FUNCTION_BLOCK fb_motorController
VAR_INPUT
	in_flg_run : BOOL;
END_VAR
VAR_OUTPUT
	out_flg_run : bool;
END_VAR
VAR
	flg_mototPowerRun: BOOL;
	flg_motorPowerReset: bool;
	fbi_delayTimerY: TON;
	fbi_delayTimerZ: TON;
	flg_rotaryPowerRun: BOOL;
	fbi_delayTimer1: TON;
END_VAR
VAR // added by the converter: edge detectors and wires of the graphical bodies
    _rt1, _rt2, _rt3, _rt4, _rt5, _rt6 : R_TRIG;
    _ft1, _ft2 : F_TRIG;
END_VAR

motorPower();
motorMoveAbs();
gm_rotary();
IF  gvl_param.var_currentMode = eP_programMode.manual OR gvl_param.var_currentMode = eP_programMode.error THEN
	motorJog();
END_IF
IF gvl_axis.axisX.NcToPlc.ActTorque > 500 THEN
	gvl_error.flg_axisXTorqueOver := TRUE;
ELSIF gvl_axis.axisY.NcToPlc.ActTorque > 500 THEN
	gvl_error.flg_axisYTorqueOver := TRUE;
ELSIF gvl_axis.axisZ.NcToPlc.ActTorque > 500 THEN
	gvl_error.flg_axisZTorqueOver := TRUE;
ELSIF gvl_axis.axisR.NcToPlc.ActTorque > 500 THEN
	gvl_error.flg_axisRTorqueOver := TRUE;
ELSE
	gvl_error.flg_axisXTorqueOver := FALSE;
	gvl_error.flg_axisYTorqueOver := FALSE;
	gvl_error.flg_axisZTorqueOver := FALSE;
	gvl_error.flg_axisRTorqueOver := FALSE;
END_IF

ACTION gm_rotary:
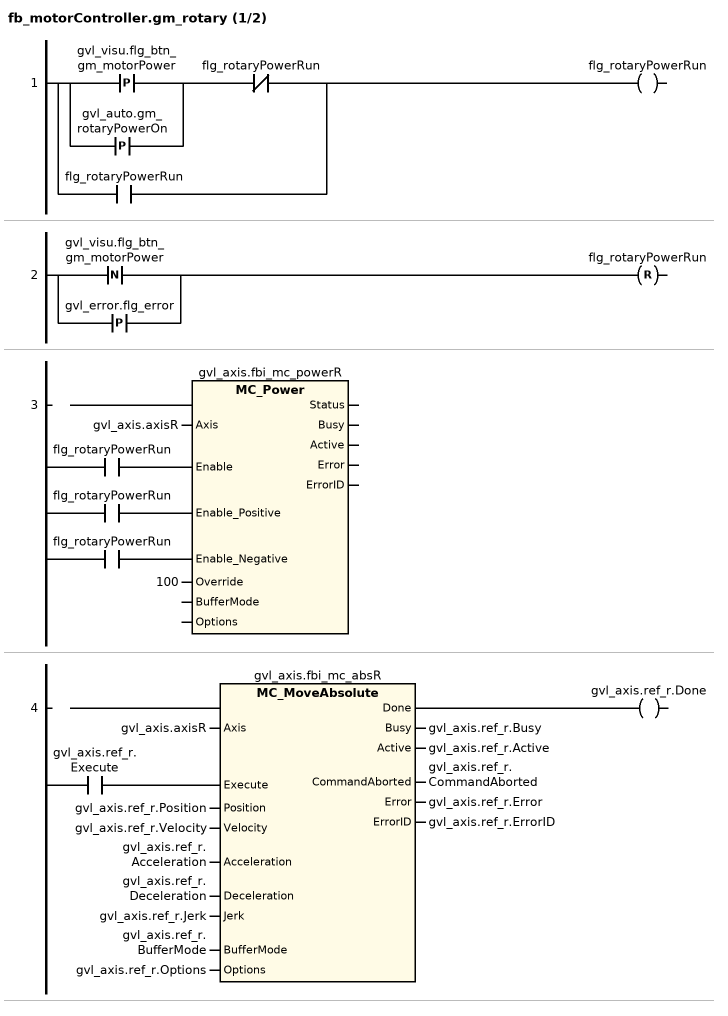
// NETWORK 1
_rt1(CLK := gvl_visu.flg_btn_gm_motorPower);
_rt2(CLK := gvl_auto.gm_rotaryPowerOn);
flg_rotaryPowerRun := (_rt1.Q OR _rt2.Q) AND NOT flg_rotaryPowerRun OR flg_rotaryPowerRun;

// NETWORK 2
_ft1(CLK := gvl_visu.flg_btn_gm_motorPower);
_rt3(CLK := gvl_error.flg_error);
flg_rotaryPowerRun R= _ft1.Q OR _rt3.Q;

// NETWORK 3
gvl_axis.fbi_mc_powerR(
    Axis := gvl_axis.axisR,
    Enable := flg_rotaryPowerRun,
    Enable_Positive := flg_rotaryPowerRun,
    Enable_Negative := flg_rotaryPowerRun,
    Override := 100); // MC_Power

// NETWORK 4
gvl_axis.fbi_mc_absR(
    Axis := gvl_axis.axisR,
    Execute := gvl_axis.ref_r.Execute,
    Position := gvl_axis.ref_r.Position,
    Velocity := gvl_axis.ref_r.Velocity,
    Acceleration := gvl_axis.ref_r.Acceleration,
    Deceleration := gvl_axis.ref_r.Deceleration,
    Jerk := gvl_axis.ref_r.Jerk,
    BufferMode := gvl_axis.ref_r.BufferMode,
    Options := gvl_axis.ref_r.Options,
    Busy => gvl_axis.ref_r.Busy,
    Active => gvl_axis.ref_r.Active,
    CommandAborted => gvl_axis.ref_r.CommandAborted,
    Error => gvl_axis.ref_r.Error,
    ErrorID => gvl_axis.ref_r.ErrorID); // MC_MoveAbsolute
gvl_axis.ref_r.Done := gvl_axis.fbi_mc_absR.Done;

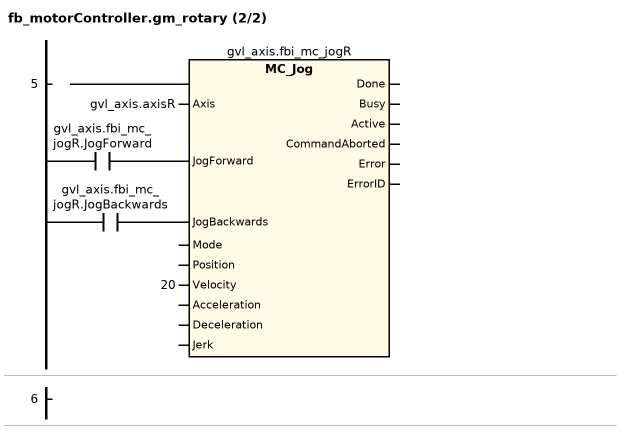
// NETWORK 5
gvl_axis.fbi_mc_jogR(
    Axis := gvl_axis.axisR,
    JogForward := gvl_axis.fbi_mc_jogR.JogForward,
    JogBackwards := gvl_axis.fbi_mc_jogR.JogBackwards,
    Velocity := 20); // MC_Jog

// NETWORK 6
END_ACTION

ACTION motorJog:
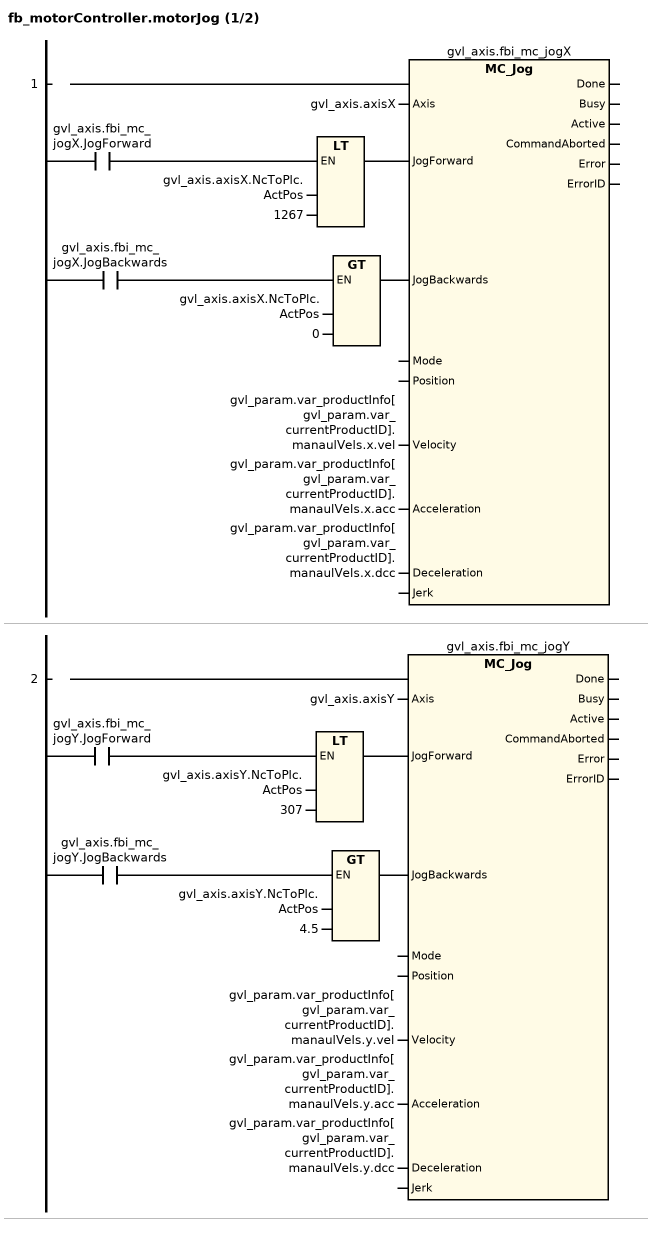
// NETWORK 1
gvl_axis.fbi_mc_jogX(
    Axis := gvl_axis.axisX,
    JogForward := gvl_axis.fbi_mc_jogX.JogForward AND gvl_axis.axisX.NcToPlc.ActPos < 1267,
    JogBackwards := gvl_axis.fbi_mc_jogX.JogBackwards AND gvl_axis.axisX.NcToPlc.ActPos > 0,
    Velocity := gvl_param.var_productInfo[gvl_param.var_currentProductID].manaulVels.x.vel,
    Acceleration := gvl_param.var_productInfo[gvl_param.var_currentProductID].manaulVels.x.acc,
    Deceleration := gvl_param.var_productInfo[gvl_param.var_currentProductID].manaulVels.x.dcc); // MC_Jog

// NETWORK 2
gvl_axis.fbi_mc_jogY(
    Axis := gvl_axis.axisY,
    JogForward := gvl_axis.fbi_mc_jogY.JogForward AND gvl_axis.axisY.NcToPlc.ActPos < 307,
    JogBackwards := gvl_axis.fbi_mc_jogY.JogBackwards AND gvl_axis.axisY.NcToPlc.ActPos > 4.5,
    Velocity := gvl_param.var_productInfo[gvl_param.var_currentProductID].manaulVels.y.vel,
    Acceleration := gvl_param.var_productInfo[gvl_param.var_currentProductID].manaulVels.y.acc,
    Deceleration := gvl_param.var_productInfo[gvl_param.var_currentProductID].manaulVels.y.dcc); // MC_Jog

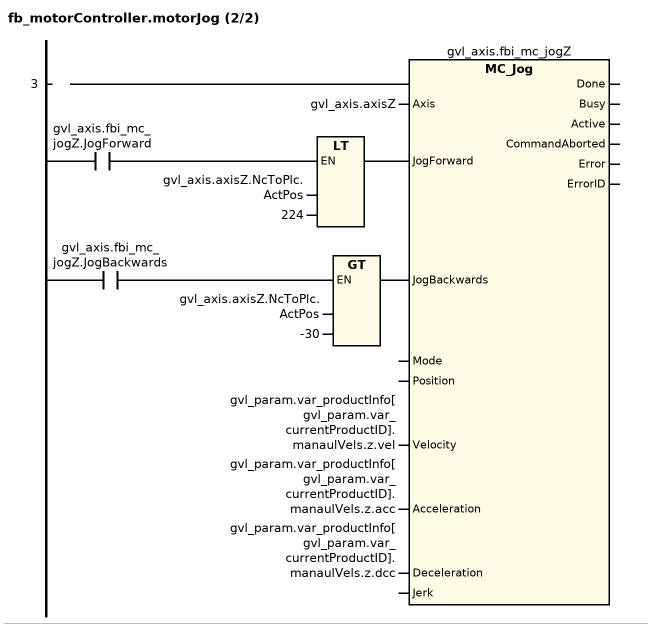
// NETWORK 3
gvl_axis.fbi_mc_jogZ(
    Axis := gvl_axis.axisZ,
    JogForward := gvl_axis.fbi_mc_jogZ.JogForward AND gvl_axis.axisZ.NcToPlc.ActPos < 224,
    JogBackwards := gvl_axis.fbi_mc_jogZ.JogBackwards AND gvl_axis.axisZ.NcToPlc.ActPos > -30,
    Velocity := gvl_param.var_productInfo[gvl_param.var_currentProductID].manaulVels.z.vel,
    Acceleration := gvl_param.var_productInfo[gvl_param.var_currentProductID].manaulVels.z.acc,
    Deceleration := gvl_param.var_productInfo[gvl_param.var_currentProductID].manaulVels.z.dcc); // MC_Jog
END_ACTION

ACTION motorMoveAbs:
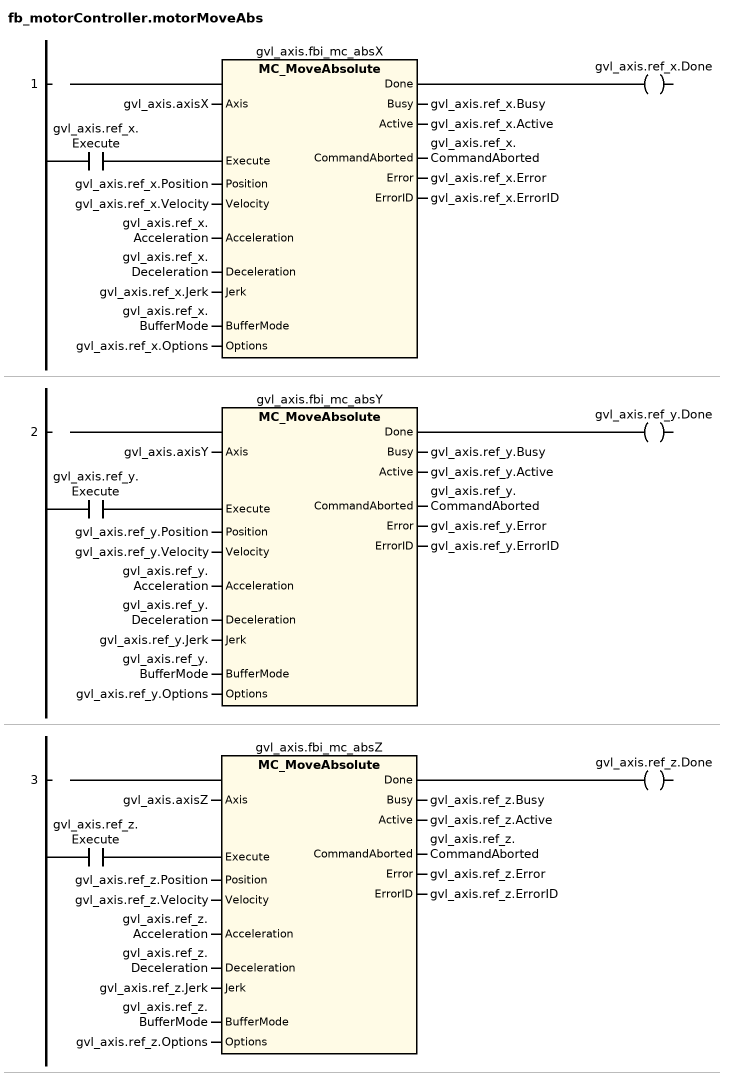
// NETWORK 1
gvl_axis.fbi_mc_absX(
    Axis := gvl_axis.axisX,
    Execute := gvl_axis.ref_x.Execute,
    Position := gvl_axis.ref_x.Position,
    Velocity := gvl_axis.ref_x.Velocity,
    Acceleration := gvl_axis.ref_x.Acceleration,
    Deceleration := gvl_axis.ref_x.Deceleration,
    Jerk := gvl_axis.ref_x.Jerk,
    BufferMode := gvl_axis.ref_x.BufferMode,
    Options := gvl_axis.ref_x.Options,
    Busy => gvl_axis.ref_x.Busy,
    Active => gvl_axis.ref_x.Active,
    CommandAborted => gvl_axis.ref_x.CommandAborted,
    Error => gvl_axis.ref_x.Error,
    ErrorID => gvl_axis.ref_x.ErrorID); // MC_MoveAbsolute
gvl_axis.ref_x.Done := gvl_axis.fbi_mc_absX.Done;

// NETWORK 2
gvl_axis.fbi_mc_absY(
    Axis := gvl_axis.axisY,
    Execute := gvl_axis.ref_y.Execute,
    Position := gvl_axis.ref_y.Position,
    Velocity := gvl_axis.ref_y.Velocity,
    Acceleration := gvl_axis.ref_y.Acceleration,
    Deceleration := gvl_axis.ref_y.Deceleration,
    Jerk := gvl_axis.ref_y.Jerk,
    BufferMode := gvl_axis.ref_y.BufferMode,
    Options := gvl_axis.ref_y.Options,
    Busy => gvl_axis.ref_y.Busy,
    Active => gvl_axis.ref_y.Active,
    CommandAborted => gvl_axis.ref_y.CommandAborted,
    Error => gvl_axis.ref_y.Error,
    ErrorID => gvl_axis.ref_y.ErrorID); // MC_MoveAbsolute
gvl_axis.ref_y.Done := gvl_axis.fbi_mc_absY.Done;

// NETWORK 3
gvl_axis.fbi_mc_absZ(
    Axis := gvl_axis.axisZ,
    Execute := gvl_axis.ref_z.Execute,
    Position := gvl_axis.ref_z.Position,
    Velocity := gvl_axis.ref_z.Velocity,
    Acceleration := gvl_axis.ref_z.Acceleration,
    Deceleration := gvl_axis.ref_z.Deceleration,
    Jerk := gvl_axis.ref_z.Jerk,
    BufferMode := gvl_axis.ref_z.BufferMode,
    Options := gvl_axis.ref_z.Options,
    Busy => gvl_axis.ref_z.Busy,
    Active => gvl_axis.ref_z.Active,
    CommandAborted => gvl_axis.ref_z.CommandAborted,
    Error => gvl_axis.ref_z.Error,
    ErrorID => gvl_axis.ref_z.ErrorID); // MC_MoveAbsolute
gvl_axis.ref_z.Done := gvl_axis.fbi_mc_absZ.Done;
END_ACTION

ACTION motorPower:
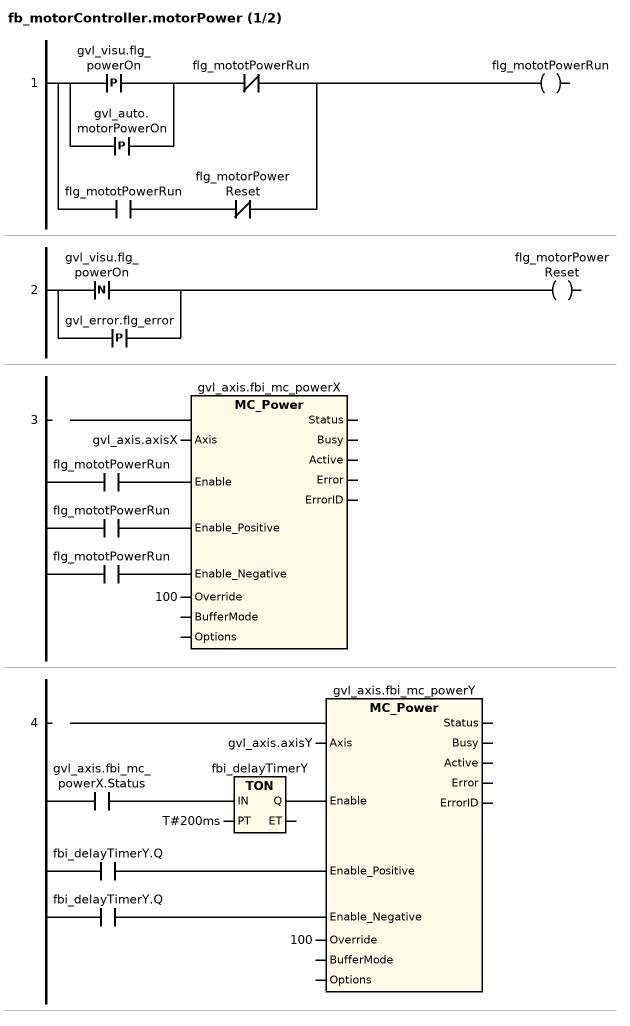
// NETWORK 1
_rt4(CLK := gvl_visu.flg_powerOn);
_rt5(CLK := gvl_auto.motorPowerOn);
flg_mototPowerRun := (_rt4.Q OR _rt5.Q) AND NOT flg_mototPowerRun OR flg_mototPowerRun AND NOT flg_motorPowerReset;

// NETWORK 2
_ft2(CLK := gvl_visu.flg_powerOn);
_rt6(CLK := gvl_error.flg_error);
flg_motorPowerReset := _ft2.Q OR _rt6.Q;

// NETWORK 3
gvl_axis.fbi_mc_powerX(
    Axis := gvl_axis.axisX,
    Enable := flg_mototPowerRun,
    Enable_Positive := flg_mototPowerRun,
    Enable_Negative := flg_mototPowerRun,
    Override := 100); // MC_Power

// NETWORK 4
fbi_delayTimerY(IN := gvl_axis.fbi_mc_powerX.Status, PT := T#200ms); // TON
gvl_axis.fbi_mc_powerY(
    Axis := gvl_axis.axisY,
    Enable := fbi_delayTimerY.Q,
    Enable_Positive := fbi_delayTimerY.Q,
    Enable_Negative := fbi_delayTimerY.Q,
    Override := 100); // MC_Power

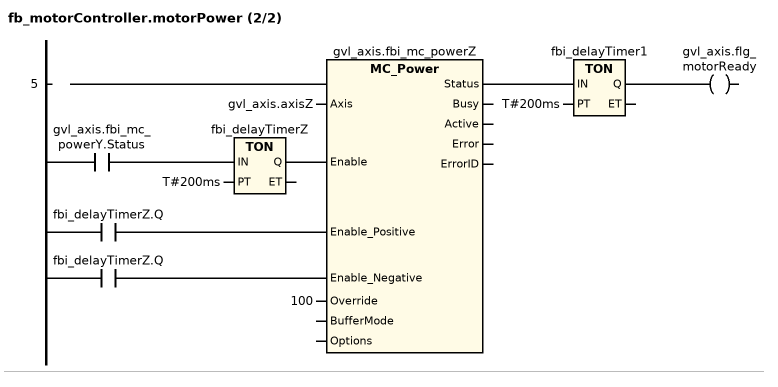
// NETWORK 5
fbi_delayTimerZ(IN := gvl_axis.fbi_mc_powerY.Status, PT := T#200ms); // TON
gvl_axis.fbi_mc_powerZ(
    Axis := gvl_axis.axisZ,
    Enable := fbi_delayTimerZ.Q,
    Enable_Positive := fbi_delayTimerZ.Q,
    Enable_Negative := fbi_delayTimerZ.Q,
    Override := 100); // MC_Power
fbi_delayTimer1(IN := gvl_axis.fbi_mc_powerZ.Status, PT := T#200ms); // TON
gvl_axis.flg_motorReady := fbi_delayTimer1.Q;
END_ACTION

END_FUNCTION_BLOCK

(* stored: Version 1.1.0.1, ProductVersion 3.1.4024.11
   POU fb_motorController: Id {a7afe743-ca97-4c0e-8d68-79cfe50368a9}, SpecialFunc None
   Action gm_rotary: Id {b7856e73-6ebc-4ae0-82c3-53629a18bb78}
   Action motorJog: Id {7593bfa0-fb25-4699-a3d8-c2b168d8aa32}
   Action motorMoveAbs: Id {aaee8c0b-c172-481b-9ed2-781416604c4a}
   Action motorPower: Id {ba9b3a69-1483-4a56-b2dd-e8174d8bc3b4} *)
